FUNCTION F_GetZonesData : ARRAY[1..NUMBER_OF_ZONES_PER_FUNCTION] OF ST_ZoneData
(**************************************************************************************
 * 	Application		:	BoxControl Framework
 *	Revision		:	$Revision: 404529 $
 *	Revision date	:	$Date: 2018-04-23 08:21:38 +0200 (Mo., 23 Apr 2018) $
 *	Last changed by	:	$Author: b7bolm $
 *	URL				:	$URL: http://almscdc.swisslog.com/repo/SWPD/Development/BoxControlFramework/20_Release/trunk/01_Software/BCF/BCF/JumpStart/20_Product/10_App/12_E_Functions/10_Lib/10_Conv/10_Functions/F_GetZonesData.TcPOU $
 *
 *	Purpose			:	Returns external zones data
 *
 * ------------------------------------------------------------------------------------
 *	Copyright Swisslog [IP AG], Switzerland. All rights reserved.
 * 
 * ------------------------------------------------------------------------------------
 *	
 * 	Revision History: 
 *
 * 	VERSION			DATE			INITIALS			DESCRIPTION
 *	0.1				01.01.2001		swl					Example
 *
 **************************************************************************************)
VAR_INPUT
	eFunctionNumber			: E_FunctionNumber; // Element function Number
END_VAR


// Check if function number is valid
IF eFunctionNumber > E_FunctionNumber.F_BEGIN_FUNCTION AND
   eFunctionNumber < E_FunctionNumber.F_END_FUNCTION THEN
  
	// Check reference is valid
	IF __ISVALIDREF(FunctionRegistry[eFunctionNumber].rFunction) THEN
   		// Return zone data
   		F_GetZonesData := FunctionRegistry[eFunctionNumber].rFunction.ZoneData;
	END_IF
END_IF

END_FUNCTION

(* stored: Version 1.1.0.1, ProductVersion 3.1.4022.12
   POU F_GetZonesData: Id {5020f816-c766-445b-9b67-fb7d1a5c6887}, SpecialFunc None *)
